FUNCTION_BLOCK fbV2_GnrStationMasterController

(*20171025 - Edit by Lim*)
(*Rung 337 - "bTransferStationBasketAvailable" variable control to solve the problem if for the basket can pick and tranfer to the same station*)


VAR_INPUT
	bTrackerEN								: BOOL;
	bTrackerBasedOnPreviousTime			: BOOL;
	bProcessCompleteBasedMasterTime		: BOOL;
	bBasketTransferCallArmInterlock			: BOOL; (* Temporary -> for GPM Only*)
	bReset									: BOOL;
	iCurrentStationAddress 					: INT;															(* Input - Define current station no so that this fb know which array number to used*)
	iPreCallArmTime							: INT;															(* Input - Pre-Call Arm Time, Program will call arm if the Total process timeEV Equal or Lesser than this value*)
	iTotalProcessTimeSV						:INT;
	iCurrentStnSeqProcessTotalTime 		: INT;															(* Input - Link with fbStnSeqProcess, to collect CurrentProcessTotalTime*)
	iPreviousStnSeqProcessTotalTime 		: INT; 															(* Input - Link with fbStnSeqProcess,  to collect PreviousProcessTotalTime*)
	iNonStopCurrentProcessTime: INT;
	bStnSeqProcessInProgressFlag			: BOOL;														(* Input - Link with fbStnSeqProcess,  to collect the status of process in progress from StnSeqProcessfb*)
	bStnSeqProcessCompleted 				: BOOL;														(* Input - Link with fbStnSeqProcess,  to collect the status of process completion from StnSeqProcessfb*)
	ARbAlternateStnEn : ARRAY [1..iAlternateSetQty] OF BOOL;
	AR2siAlternateStn : ARRAY [1..iAlternateSetQty, 1..iAlternateStnQty] OF INT;
(*	DSStnSeqProOutput 				:DS_StnSeqProOutput;								(* Output - To Control Output - When process running, instrument should control by the output in this Data structure*)
*)

END_VAR

VAR_IN_OUT PERSISTENT
	bStnSeqProcessSt						: BOOL;														(* Output - Link with fbStnSeqProcess, After Read out from fbGnrProductRecipeMemory, this fb will trigger this Bool to start the StnSeqProcess*)

	ARbProductRecipeCallEn 				: ARRAY [0..iStnQty] OF BOOL;					(* Output - Link with fbGnrProductRecipeMemory, Array based on Current Station No, the fbGnrProductRecipeMemory will start Read info from Memory when this bool turn on*)
	ARiProductRecipeNoCall 				: ARRAY [0..iStnQty] OF INT;						(* Output - Link with fbGnrProductRecipeMemory, Array based on Current Station No, the read out from fbGnrProductRecipeMemory is based on this Product Recipe No*)
	ARiProductRecipeStepCall 				: ARRAY [0..iStnQty] OF INT;						(* Output - Link with fbGnrProductRecipeMemory, Array based on Current Station No, the read out from fbGnrProductRecipeMemory is based on this Product Recipe Step No*)
	DSfbGnrProductRecipeMemoryOut 		: DSV2_fbGnrProductRecipeMemoryOut;						(* Input - Link with fbGnrProductRecipeMemory, all the read out info from fbGnrProductRecipeMemory will store in this DataStucture*)

	ARbArmReady						: ARRAY [1..iArmQty] OF BOOL;								(* Input - From ArmPnpFB, This signal is used to confirm if the arm is ready and idling*)
	ARiStnNoToCalledArm					: ARRAY [0..iArmQty] OF INT; 									(* Output - Link with fbArmPnP, Array based on Arm No, The Int will store which Station that calling the Arm*)
	ARDSGnrFeedArmPnpParameter		: ARRAY [0..iArmQty] OF DSV2_Gnr_CalledArmPnpParameter; 	(* Output - Link with fbArmPnP, Array based on Current Station No, Arm should move based on this DataStructure Info*)

	ARDSLdBasketInfo		 				: ARRAY [0..iLdStnQty] OF DSV2_BasketInfo;								(*Input - Loading CONFIRM Basket Info*)
	ARDSUldBasketInfo		 				: ARRAY [0..iUldStnQty] OF DSV2_BasketInfo;							(*Input - Uloading CONFIRM Basket Info*)
	ARDsStnBasketInfo					: ARRAY [0..iStnQty] OF DSV2_BasketInfo;									(*Input - Station Basket Info*)


END_VAR

VAR_OUTPUT PERSISTENT

	DSGnrBufferCalledArmPnpParameter 	: DSV2_Gnr_CalledArmPnpParameter;							(* Internal used, Buffer Data Structure read out from fbGnrProductRecipeMemory*)
	DSGnrBuffersPnpSequenceDescription	: STRING (99);													(* Internal used, Buffer Description read out from fbGnrProductRecipeMemory*)
	ARiPreviousStnSeqTotalProcessTime 	: ARRAY [0..iProductRecipeArrayQty] OF INT;				(* Internal used, Previous Total Process Time will save into this Array, Array based on StationSequenceNo*)
	iMasterTimeCallArmCountDownTime: INT;
	iMasterTimeBasedProcessCompleteFlag : BOOL;
	iCallStep									: INT;															(* Internal used, to monitor the current Step so that you can indentify the error of this function block if stucked*)

END_VAR
VAR PERSISTENT
	DSfbGnrProductRecipeMemoryOutErrorLog 		: DSV2_fbGnrProductRecipeMemoryOut;
	DSCurrentStationBasketInfoErrorLog				: DSV2_BasketInfo;

	bBasketDetectedRE						: R_TRIG;
	iCallCheck								: INT;
	bArmPnpSequenceCallEn				: BOOL;
	bStnSeqProcessCompletedRE			: R_TRIG;
	iCallArmCountDownTime				: INT;
	bCallArmEnInt								: BOOL;


END_VAR
VAR
	bBasketDetectedFE						: F_TRIG;
	bCallProductRecipeStorageEn			: BOOL;
	bTestCallArm								: BOOL;

	DSCurrentStationBasketInfo: DSV2_BasketInfo;
	DSEmptyBasketInfo: DSV2_BasketInfo;
	bPickStationBasketAvailable: BOOL;
	bTransferStationBasketAvailable: BOOL;
	bTransferStationBasketNotAvailable: BOOL;
	iCurrentStationAddressInt: INT;
	iTrackerCallArmCountDownTime: INT;
(*	bAlternateStnEnableFound: BOOL;*)
(*	iCheckAlternateStnEnFL: INT;*)
	bPickAltStnIDFound: BOOL;
	iPickAlternateStnFindFL: INT;
	iPickAlternateSetFindFL: INT;
	iPickAltStnTransferFL : INT;
	ARiBufferPickAltStn: ARRAY [1..iAlternateStnQty] OF INT;

	bTransferAltStnIDFound: BOOL;
	iTransferAlternateStnFindFL: INT;
	iTransferAlternateSetFindFL: INT;
	iTransferAltStnTransferFL : INT;
	ARiBufferTransferAltStn: ARRAY [1..iAlternateStnQty] OF INT;

	iCheckTrfStnBktFL: INT;
	iTransferStnNo: INT;
	iAltTransferStnNo: INT;
	iSearchLdStnFL: INT;
	bLdStnFound: BOOL;
	iSearchStnIDFL: INT;
	iSearchStnIDFound: BOOL;
	DSUldBasketInfo: BOOL;
	iSearchLdStnIDFound: BOOL;
	iSearchUldStnIDFound: BOOL;
	iCheckTrfStnBktSFL: INT;
	bReadyToCallArm: BOOL;
	bTrackerBasedPreviousTimeCallArm: BOOL;
	bTrackerNotBasedPreviousTimeCallArm: BOOL;
	bDataInBufferCalledArmPnpParameterDone: BOOL;
	bResetRE: R_TRIG;
	tErrorLoopingTimer: TON;
END_VAR

bResetRE(CLK:=bReset , Q=> );


(*Check if Loading Stn Detected, Switch the CurrentStatonAddress to 0*)
bLdStnFound:=FALSE;
iSearchLdStnFL := 1;
	FOR iSearchLdStnFL := 1 TO iLdStnQty DO
		IF iSearchLdStnFL >= 1 AND iSearchLdStnFL <= iLdStnQty THEN
			IF ARiLdStnID[iSearchLdStnFL] = iCurrentStationAddress THEN
			iCurrentStationAddressInt := 0;
			bLdStnFound:=TRUE;
			END_IF
		END_IF
	END_FOR

IF NOT bLdStnFound THEN
iCurrentStationAddressInt := iCurrentStationAddress;
END_IF


(*Check if Alternate Stn Matched with Current (Pick) Station*)
bPickAltStnIDFound := FALSE;
iPickAlternateSetFindFL := 1;
	FOR iPickAlternateSetFindFL := 1 TO iAlternateSetQty DO
		IF iPickAlternateSetFindFL >= 1 AND iPickAlternateSetFindFL <= iAlternateSetQty THEN
			IF ARbAlternateStnEn[iPickAlternateSetFindFL] THEN
			iPickAlternateStnFindFL := 1; (*Find Stn ID matching*)
				FOR iPickAlternateStnFindFL := 1 TO iAlternateStnQty DO
					IF iPickAlternateStnFindFL >= 1 AND iPickAlternateStnFindFL <= iAlternateStnQty THEN
						IF iCurrentStationAddress = AR2SiAlternateStn[iPickAlternateSetFindFL , iPickAlternateStnFindFL] THEN
							bPickAltStnIDFound := TRUE;
							iPickAltStnTransferFL := 1;
								FOR iPickAltStnTransferFL := 1 TO iAlternateStnQty DO
									IF iPickAltStnTransferFL >= 1 AND iPickAltStnTransferFL <= iAlternateStnQty THEN
										ARiBufferPickAltStn[iPickAltStnTransferFL] := AR2SiAlternateStn[iPickAlternateSetFindFL , iPickAltStnTransferFL];
									END_IF
								END_FOR
							iPickAlternateSetFindFL := iAlternateSetQty+1;
							iPickAlternateStnFindFL := iAlternateStnQty+1;
							iPickAltStnTransferFL := iAlternateStnQty+1;

						END_IF
					END_IF
				END_FOR
			END_IF
		END_IF
	END_FOR

(*Check if Alternate Stn Matched with Transfer Station*)

bTransferAltStnIDFound := FALSE;
IF iCallStep = 3 THEN
iTransferAlternateSetFindFL := 1;
	FOR iTransferAlternateSetFindFL := 1 TO iAlternateSetQty DO
		IF iTransferAlternateSetFindFL >= 1 AND iTransferAlternateSetFindFL <= iAlternateSetQty THEN
			IF ARbAlternateStnEn[iTransferAlternateSetFindFL] THEN
			iTransferAlternateStnFindFL := 1; (*Find Stn ID matching*)
				FOR iTransferAlternateStnFindFL := 1 TO iAlternateStnQty DO
					IF iTransferAlternateStnFindFL >= 1 AND iTransferAlternateStnFindFL <= iAlternateStnQty THEN
						IF DSGnrBufferCalledArmPnpParameter.iTransferStationNo = AR2SiAlternateStn[iTransferAlternateSetFindFL , iTransferAlternateStnFindFL] THEN
							bTransferAltStnIDFound := TRUE;
							iTransferAltStnTransferFL := 1;
								FOR iTransferAltStnTransferFL := 1 TO iAlternateStnQty DO
									IF iTransferAltStnTransferFL >= 1 AND iTransferAltStnTransferFL <= iAlternateStnQty THEN
										ARiBufferTransferAltStn[iTransferAltStnTransferFL] := AR2SiAlternateStn[iTransferAlternateSetFindFL , iTransferAltStnTransferFL];
									END_IF
								END_FOR
							iTransferAlternateSetFindFL := iAlternateSetQty+1;
							iTransferAlternateStnFindFL := iAlternateStnQty+1;
							iTransferAltStnTransferFL := iAlternateStnQty+1;

						END_IF
					END_IF
				END_FOR
			END_IF
		END_IF
	END_FOR
END_IF

(*Define Current Station Basket Info*)
iSearchLdStnIDFound := FALSE;
iSearchUldStnIDFound := FALSE;


IF NOT iSearchLdStnIDFound AND NOT iSearchUldStnIDFound THEN
	iSearchStnIDFL := 1;
		FOR iSearchStnIDFL := 1 TO iLdStnQty DO
			IF iSearchStnIDFL >= 1 AND iSearchStnIDFL <= iLdStnQty THEN
				IF iCurrentStationAddress = ARiLdStnID[iSearchStnIDFL] THEN
					DSCurrentStationBasketInfo := ARDSLdBasketInfo[iSearchStnIDFL];
					iSearchLdStnIDFound := TRUE;
				END_IF
			END_IF
		END_FOR
END_IF


IF NOT iSearchLdStnIDFound AND NOT iSearchUldStnIDFound THEN
	iSearchStnIDFL := 1;
		FOR iSearchStnIDFL := 1 TO iUldStnQty DO
			IF iSearchStnIDFL >= 1 AND iSearchStnIDFL <= iUldStnQty THEN
				IF iCurrentStationAddress = ARiUldStnID[iSearchStnIDFL] THEN
					DSCurrentStationBasketInfo := ARDSUldBasketInfo[iSearchStnIDFL];
					iSearchUldStnIDFound := TRUE;
				END_IF
			END_IF
		END_FOR
END_IF


IF NOT iSearchLdStnIDFound AND NOT iSearchUldStnIDFound THEN
	IF iCurrentStationAddress >= 1 AND iCurrentStationAddress <= iStnQty THEN
	DSCurrentStationBasketInfo := ARDsStnBasketInfo[iCurrentStationAddress];
	ELSE
	DSCurrentStationBasketInfo := DSEmptyBasketInfo;
	END_IF
END_IF


(* Check if no one called Data From DSfbGnrProductRecipeMemory *)
iCallCheck := 1;
FOR iCallCheck := 1 TO iStnQty DO
		IF ARbProductRecipeCallEn[iCallCheck] THEN
		bArmPnpSequenceCallEn := TRUE;
		iCallCheck := 90;
		END_IF
END_FOR

IF iCallCheck > iStnQty AND iCallCheck <= (iStnQty+2) THEN
bArmPnpSequenceCallEn := FALSE;
END_IF


(*[][][][][][][][][][][][][][][][][][][][][][][][][][][][][][][][][][][][][][][][][][][][][][][][][][][][][][][][][][][][][][][][][][][][][][][][][][][][][][][][][][][][][][][][][][][][][][][][][][][]*)
(*Store Previous Total Process Time by Program No*)
bStnSeqProcessCompletedRE(CLK:=bStnSeqProcessCompleted , Q=> );

IF bStnSeqProcessCompletedRE.Q AND (*ARiPreviousStnSeqTotalProcessTime[*)DSCurrentStationBasketInfo.iStationSeqenceRecipeNo(*]*) > 0
AND (*ARiPreviousStnSeqTotalProcessTime[*)DSCurrentStationBasketInfo.iStationSeqenceRecipeNo(*]*) <= iProductRecipeArrayQty THEN
ARiPreviousStnSeqTotalProcessTime[DSCurrentStationBasketInfo.iStationSeqenceRecipeNo] := iPreviousStnSeqProcessTotalTime ;
END_IF


(*[][][][][][][][][][][][][][][][][][][][][][][][][][][][][][][][][][][][][][][][][][][][][][][][][][][][][][][][][][][][][][][][][][][][][][][][][][][][][][][][][][][][][][][][][][][][][][][][][][][]*)
(*Call Arm Activation*)

IF (*NOT DSStnSeqProOutput.b12SlowPull AND*) (bStnSeqProcessInProgressFlag OR bStnSeqProcessCompleted) THEN
	iCallArmCountDownTime := ARiPreviousStnSeqTotalProcessTime[DSCurrentStationBasketInfo.iStationSeqenceRecipeNo] - iCurrentStnSeqProcessTotalTime;
	iMasterTimeCallArmCountDownTime := iTotalProcessTimeSV - iNonStopCurrentProcessTime;
ELSE
(*LKT added 170321*)
 	iCallArmCountDownTime := 0;
	iMasterTimeCallArmCountDownTime := 0;


END_IF

IF iMasterTimeCallArmCountDownTime <= 0 AND bDataInBufferCalledArmPnpParameterDone THEN
iMasterTimeBasedProcessCompleteFlag := TRUE;
ELSE
iMasterTimeBasedProcessCompleteFlag := FALSE;
END_IF

(*
IF DSStnSeqProOutput.b12SlowPull AND bStnSeqProcessInProgressFlag OR bStnSeqProcessCompleted THEN
	iCallArmCountDownTime := iTotalProcessTimeSV - iCurrentStnSeqProcessTotalTime;
END_IF
*)

iTrackerCallArmCountDownTime := iTotalProcessTimeSV - iCurrentStnSeqProcessTotalTime;

IF NOT bProcessCompleteBasedMasterTime AND
(NOT iSearchLdStnIDFound AND NOT bTrackerEN  AND iCurrentStnSeqProcessTotalTime > 0 AND iCallArmCountDownTime >= 0 AND iCallArmCountDownTime <= iPreCallArmTime AND bStnSeqProcessInProgressFlag) THEN
bReadyToCallArm := TRUE;
ELSIF bProcessCompleteBasedMasterTime AND
(NOT iSearchLdStnIDFound AND NOT bTrackerEN  AND iNonStopCurrentProcessTime > 0 AND iTotalProcessTimeSV >= 0 AND iMasterTimeCallArmCountDownTime <= iPreCallArmTime AND (bStnSeqProcessInProgressFlag OR bStnSeqProcessCompleted) )THEN
bReadyToCallArm := TRUE;
ELSE
bReadyToCallArm := FALSE;
END_IF

IF NOT bProcessCompleteBasedMasterTime AND
(NOT iSearchLdStnIDFound  AND bTrackerEN AND bTrackerBasedOnPreviousTime  AND iCurrentStnSeqProcessTotalTime > 0 AND iCallArmCountDownTime >= 0 AND iCallArmCountDownTime <= iPreCallArmTime AND bStnSeqProcessInProgressFlag) THEN
bReadyToCallArm := TRUE;
ELSIF bProcessCompleteBasedMasterTime AND
(NOT iSearchLdStnIDFound  AND bTrackerEN AND bTrackerBasedOnPreviousTime  AND iNonStopCurrentProcessTime > 0 AND iTotalProcessTimeSV >= 0 AND iMasterTimeCallArmCountDownTime <= iPreCallArmTime AND (bStnSeqProcessInProgressFlag OR bStnSeqProcessCompleted)) THEN
bTrackerBasedPreviousTimeCallArm := TRUE;
ELSE
bTrackerBasedPreviousTimeCallArm := FALSE;
END_IF


IF NOT bProcessCompleteBasedMasterTime AND
(NOT iSearchLdStnIDFound AND bTrackerEN AND NOT bTrackerBasedOnPreviousTime AND iCurrentStnSeqProcessTotalTime > 0 AND iTrackerCallArmCountDownTime >= 0 AND iTrackerCallArmCountDownTime <= iPreCallArmTime AND bStnSeqProcessInProgressFlag) THEN
bReadyToCallArm := TRUE;
ELSIF bProcessCompleteBasedMasterTime AND
(NOT iSearchLdStnIDFound AND bTrackerEN AND NOT bTrackerBasedOnPreviousTime AND iNonStopCurrentProcessTime > 0 AND iTotalProcessTimeSV >= 0 AND iMasterTimeCallArmCountDownTime <= iPreCallArmTime AND  (bStnSeqProcessInProgressFlag OR bStnSeqProcessCompleted)) THEN
bTrackerNotBasedPreviousTimeCallArm := TRUE;
ELSE
bTrackerNotBasedPreviousTimeCallArm := FALSE;
END_IF




IF bReadyToCallArm
OR
bTrackerBasedPreviousTimeCallArm
OR
bTrackerNotBasedPreviousTimeCallArm
OR
(iSearchLdStnIDFound AND bStnSeqProcessCompleted)
OR
bTestCallArm
THEN
bCallArmEnInt := TRUE;
ELSE
bCallArmEnInt := FALSE;
END_IF

(*Check PickStation Basket Availability *)
IF (*DSGnrBufferCalledArmPnpParameter.iPickStationNo*)iSearchLdStnIDFound AND DSCurrentStationBasketInfo.bAvailibility THEN
bPickStationBasketAvailable := TRUE;
ELSIF (*DSGnrBufferCalledArmPnpParameter.iPickStationNo*)iSearchUldStnIDFound AND DSCurrentStationBasketInfo.bAvailibility THEN
bPickStationBasketAvailable := TRUE;
ELSIF (*DSGnrBufferCalledArmPnpParameter.iPickStationNo*)iCurrentStationAddress >= 1 AND  (*DSGnrBufferCalledArmPnpParameter.iPickStationNo*)iCurrentStationAddress <= iStnQty AND ARDsStnBasketInfo[(*DSGnrBufferCalledArmPnpParameter.iPickStationNo*)iCurrentStationAddress].bAvailibility THEN
bPickStationBasketAvailable := TRUE;
ELSE
bPickStationBasketAvailable := FALSE;
END_IF
(*
(*Check TransferStation Basket Availability *)
IF DSGnrBufferCalledArmPnpParameter.iTransferStationNo = ARiLdStnID AND DSLdBasketInfo.bAvailibility THEN
bTransferStationBasketAvailable := TRUE;
ELSIF DSGnrBufferCalledArmPnpParameter.iTransferStationNo = ARiUldStnID AND DSUldBasketInfo.bAvailibility THEN
bTransferStationBasketAvailable := TRUE;
ELSIF DSGnrBufferCalledArmPnpParameter.iTransferStationNo >= 1 AND  DSGnrBufferCalledArmPnpParameter.iTransferStationNo <= iStnQty AND ARDsStnBasketInfo[DSGnrBufferCalledArmPnpParameter.iTransferStationNo].bAvailibility THEN
bTransferStationBasketAvailable := TRUE;
ELSE
bTransferStationBasketAvailable := FALSE;
END_IF
*)

IF bTransferAltStnIDFound THEN
	iCheckTrfStnBktFL := 1;
	bTransferStationBasketAvailable := TRUE;
	iAltTransferStnNo := 0;
	FOR iCheckTrfStnBktFL := 1 TO iAlternateStnQty DO

		IF iCheckTrfStnBktFL >= 1 AND iCheckTrfStnBktFL <= iAlternateStnQty THEN

			IF bTransferStationBasketAvailable THEN
			iCheckTrfStnBktSFL := 1;
				FOR iCheckTrfStnBktSFL := 1 TO iLdStnQty DO
					IF iCheckTrfStnBktSFL >= 1 AND iCheckTrfStnBktSFL <= iLdStnQty THEN

						IF ARiBufferTransferAltStn[iCheckTrfStnBktFL] = ARiLdStnID[iCheckTrfStnBktSFL] AND NOT ARDSLdBasketInfo[iCheckTrfStnBktSFL].bAvailibility THEN
						bTransferStationBasketAvailable := FALSE;
						iAltTransferStnNo := ARiBufferTransferAltStn[iCheckTrfStnBktFL];
						iCheckTrfStnBktFL := iAlternateStnQty+1;
						END_IF
					END_IF
				END_FOR
			END_IF


			IF bTransferStationBasketAvailable THEN
			iCheckTrfStnBktSFL := 1;
				FOR iCheckTrfStnBktSFL := 1 TO iUldStnQty DO
					IF iCheckTrfStnBktSFL >= 1 AND iCheckTrfStnBktSFL <= iUldStnQty THEN

						IF ARiBufferTransferAltStn[iCheckTrfStnBktFL] = ARiUldStnID[iCheckTrfStnBktSFL] AND NOT ARDSUldBasketInfo[iCheckTrfStnBktSFL].bAvailibility THEN
						bTransferStationBasketAvailable := FALSE;
						iAltTransferStnNo := ARiBufferTransferAltStn[iCheckTrfStnBktFL];
						iCheckTrfStnBktFL := iAlternateStnQty+1;
						END_IF
					END_IF
				END_FOR
			END_IF


			IF bTransferStationBasketAvailable AND  ARiBufferTransferAltStn[iCheckTrfStnBktFL] >= 1 AND ARiBufferTransferAltStn[iCheckTrfStnBktFL] <= iStnQty AND NOT  ARDsStnBasketInfo[ARiBufferTransferAltStn[iCheckTrfStnBktFL]].bAvailibility THEN
			bTransferStationBasketAvailable := FALSE;
			iAltTransferStnNo := ARiBufferTransferAltStn[iCheckTrfStnBktFL];
			iCheckTrfStnBktFL := iAlternateStnQty+1;

			END_IF

			(*To solve the problem if for the basket can pick and tranfer to the same station*)
			IF iCurrentStationAddress = DSGnrBufferCalledArmPnpParameter.iTransferStationNo THEN
			bTransferStationBasketAvailable := FALSE;
			iAltTransferStnNo := DSGnrBufferCalledArmPnpParameter.iTransferStationNo;
			iCheckTrfStnBktFL := iAlternateStnQty+1;

			END_IF



		END_IF

	END_FOR

ELSE

	bTransferStationBasketAvailable := FALSE;
	
	IF NOT bTransferStationBasketAvailable THEN
	iCheckTrfStnBktSFL := 1;
		FOR iCheckTrfStnBktSFL := 1 TO iLdStnQty DO
			IF iCheckTrfStnBktSFL >= 1 AND iCheckTrfStnBktSFL <= iLdStnQty THEN
				IF DSGnrBufferCalledArmPnpParameter.iTransferStationNo = ARiLdStnID[iCheckTrfStnBktSFL] AND ARDSLdBasketInfo[iCheckTrfStnBktSFL].bAvailibility THEN
					bTransferStationBasketAvailable := TRUE;
				END_IF
			END_IF
		END_FOR
	END_IF
	
	
	IF NOT bTransferStationBasketAvailable THEN
	iCheckTrfStnBktSFL := 1;
		FOR iCheckTrfStnBktSFL := 1 TO iUldStnQty DO
			IF iCheckTrfStnBktSFL >= 1 AND iCheckTrfStnBktSFL <= iUldStnQty THEN
				IF DSGnrBufferCalledArmPnpParameter.iTransferStationNo = ARiUldStnID[iCheckTrfStnBktSFL] AND ARDSUldBasketInfo[iCheckTrfStnBktSFL].bAvailibility THEN
				bTransferStationBasketAvailable := TRUE;
				END_IF
			END_IF
		END_FOR
	END_IF
	
	
	IF NOT bTransferStationBasketAvailable THEN
		IF DSGnrBufferCalledArmPnpParameter.iTransferStationNo >= 1 AND  DSGnrBufferCalledArmPnpParameter.iTransferStationNo <= iStnQty AND ARDsStnBasketInfo[DSGnrBufferCalledArmPnpParameter.iTransferStationNo].bAvailibility THEN
			bTransferStationBasketAvailable := TRUE;
		END_IF
	END_IF

	(*To solve the problem if for the basket can pick and tranfer to the same station*)
	IF iCurrentStationAddress = DSGnrBufferCalledArmPnpParameter.iTransferStationNo THEN
	bTransferStationBasketAvailable := FALSE;
	END_IF


END_IF

IF bCallArmEnInt
AND bBasketTransferCallArmInterlock (*To be delete, This interlock for GPM Johor Only*)
AND bPickStationBasketAvailable
AND NOT bTransferStationBasketAvailable
AND ARbArmReady[DSGnrBufferCalledArmPnpParameter.iCallArmNo]
AND  ARiStnNoToCalledArm[DSGnrBufferCalledArmPnpParameter.iCallArmNo] = 0
AND iCallStep = 3
THEN

	IF bTransferAltStnIDFound THEN
		ARDSGnrFeedArmPnpParameter[DSGnrBufferCalledArmPnpParameter.iCallArmNo] := DSGnrBufferCalledArmPnpParameter;
		ARDSGnrFeedArmPnpParameter[DSGnrBufferCalledArmPnpParameter.iCallArmNo].iPickStationNo := iCurrentStationAddress;
		ARDSGnrFeedArmPnpParameter[DSGnrBufferCalledArmPnpParameter.iCallArmNo].iTransferStationNo := iAltTransferStnNo;

		ARiStnNoToCalledArm[DSGnrBufferCalledArmPnpParameter.iCallArmNo]  := iCurrentStationAddress;

	ELSE

		ARDSGnrFeedArmPnpParameter[DSGnrBufferCalledArmPnpParameter.iCallArmNo] := DSGnrBufferCalledArmPnpParameter;
		ARDSGnrFeedArmPnpParameter[DSGnrBufferCalledArmPnpParameter.iCallArmNo].iPickStationNo := iCurrentStationAddress;
		ARiStnNoToCalledArm[DSGnrBufferCalledArmPnpParameter.iCallArmNo]  := iCurrentStationAddress;

	END_IF

bDataInBufferCalledArmPnpParameterDone := TRUE;

END_IF

IF NOT bCallArmEnInt THEN
bDataInBufferCalledArmPnpParameterDone := FALSE;
END_IF


(*[][][][][][][][][][][][][][][][][][][][][][][][][][][][][][][][][][][][][][][][][][][][][][][][][][][][][][][][][][][][][][][][][][][][][][][][][][][][][][][][][][][][][][][][][][][][][][][][][][][]*)
(*Start Call *)
bBasketDetectedRE(CLK:=DSCurrentStationBasketInfo.bAvailibility , Q=> );
bBasketDetectedFE(CLK:=DSCurrentStationBasketInfo.bAvailibility , Q=> );
(*
IF bBasketDetectedRE.Q THEN
DSCurrentStationBasketInfo.iStationSeqenceRecipeNo :=  0;
END_IF
*)
IF DSCurrentStationBasketInfo.bAvailibility AND NOT bReset AND NOT bCallProductRecipeStorageEn AND NOT bArmPnpSequenceCallEn THEN
ARbProductRecipeCallEn[iCurrentStationAddressInt] := TRUE;
iCallStep := 1;
bCallProductRecipeStorageEn := TRUE;
END_IF

IF DSCurrentStationBasketInfo.bAvailibility AND DSCurrentStationBasketInfo.iStationSeqenceRecipeNo > 0 THEN (*New, Make sure during ArmPnP, must write the StnSeqRecipeNo to BasketInfo before put the basket to station*)
bStnSeqProcessSt := TRUE;
ELSE
bStnSeqProcessSt := FALSE;
END_IF


(*Error Looping Control*)
tErrorLoopingTimer(IN:=iCallStep = 11 OR iCallStep = 12 , PT:=t#3s , Q=> , ET=> );

	IF tErrorLoopingTimer.Q THEN
	bCallProductRecipeStorageEn := FALSE;
	iCallStep := 0;
	END_IF

IF bBasketDetectedFE.Q OR bResetRE.Q THEN
iCallStep := 0;
END_IF



CASE iCallStep OF

0:
ARbProductRecipeCallEn[iCurrentStationAddressInt] := FALSE;
ARiProductRecipeNoCall[iCurrentStationAddressInt] := 0;
ARiProductRecipeStepCall[iCurrentStationAddressInt] := 0;

bCallProductRecipeStorageEn := FALSE;
bStnSeqProcessSt := FALSE;


1:

ARiProductRecipeNoCall[iCurrentStationAddressInt] := DSCurrentStationBasketInfo.iProductRecipeNo;
ARiProductRecipeStepCall[iCurrentStationAddressInt] := DSCurrentStationBasketInfo.iProductRecipeStepNo+1(*New*);
ARbProductRecipeCallEn[iCurrentStationAddressInt] := TRUE;
iCallStep := 2;

2:

IF DSfbGnrProductRecipeMemoryOut.bCallCompleted
AND  DSfbGnrProductRecipeMemoryOut.iCalledProductRecipeNo = DSCurrentStationBasketInfo.iProductRecipeNo
AND DSfbGnrProductRecipeMemoryOut.iCalledProductRecipeStep = DSCurrentStationBasketInfo.iProductRecipeStepNo+1(*New*)
AND NOT DSfbGnrProductRecipeMemoryOut.bCallPickStationNoErr
AND NOT DSfbGnrProductRecipeMemoryOut.bCallTransferStationNoErr
AND NOT DSfbGnrProductRecipeMemoryOut.bCallUpDownPatternMemoryErr
AND NOT DSfbGnrProductRecipeMemoryOut.bInvalidProductRecipeNoErrHold
AND NOT DSfbGnrProductRecipeMemoryOut.bInvalidProductRecipeNoErrPulse
AND NOT DSfbGnrProductRecipeMemoryOut.bInvalidProductRecipeStepErrHold
AND NOT DSfbGnrProductRecipeMemoryOut.bInvalidProductRecipeStepErrPulse
THEN

DSGnrBufferCalledArmPnpParameter := DSfbGnrProductRecipeMemoryOut.DSGnrCalledArmPnpParameter;
DSGnrBuffersPnpSequenceDescription := DSfbGnrProductRecipeMemoryOut.sProductRecipeDescription;
(*DSCurrentStationBasketInfo.iStationSeqenceRecipeNo := DSGnrBufferCalledArmPnpParameter.iStnSeqRecipeNo;*) (*New*)
ARbProductRecipeCallEn[iCurrentStationAddressInt] := FALSE;
iCallStep := 3;
END_IF

IF DSfbGnrProductRecipeMemoryOut.bCallCompleted
AND (  DSfbGnrProductRecipeMemoryOut.iCalledProductRecipeNo <> DSCurrentStationBasketInfo.iProductRecipeNo
OR DSfbGnrProductRecipeMemoryOut.iCalledProductRecipeStep <> DSCurrentStationBasketInfo.iProductRecipeStepNo+1(*New*))
THEN
ARbProductRecipeCallEn[iCurrentStationAddressInt] := FALSE;
iCallStep := 11;
END_IF


IF DSfbGnrProductRecipeMemoryOut.bCallCompleted
AND (DSfbGnrProductRecipeMemoryOut.bCallPickStationNoErr
OR DSfbGnrProductRecipeMemoryOut.bCallTransferStationNoErr
OR DSfbGnrProductRecipeMemoryOut.bCallUpDownPatternMemoryErr
OR DSfbGnrProductRecipeMemoryOut.bInvalidProductRecipeNoErrHold
OR DSfbGnrProductRecipeMemoryOut.bInvalidProductRecipeNoErrPulse
OR DSfbGnrProductRecipeMemoryOut.bInvalidProductRecipeStepErrHold
OR DSfbGnrProductRecipeMemoryOut.bInvalidProductRecipeStepErrPulse)
THEN
ARbProductRecipeCallEn[iCurrentStationAddressInt] := FALSE;
iCallStep := 12;
END_IF

3: (*Complete without Error*);
ARbProductRecipeCallEn[iCurrentStationAddressInt] := FALSE;


11: (*Program No or Step No Not Matching*);



12: (*Error when call data *);

END_CASE


(*[][][][][][][][][][][][][][][][][][][][][][][][][][][][][][][][][][][][][][][][][][][][][][][][][][][][][][][][][][][][][][][][][][][][][][][][][][][][][][][][][][][][][][][][][][][][][][][][][][][]*)

END_FUNCTION_BLOCK

(* stored: Version 1.1.0.1, ProductVersion 3.1.4024.12
   POU fbV2_GnrStationMasterController: Id {a3ca15e1-e95b-481a-a44e-f455bbe104e2}, SpecialFunc None *)
